// TIA Portal V20 export
VAR_GLOBAL   // PLC tag table "Inputs"
   "Switch 1 ON" AT %I16.0 : Bool;
   "Switch 2 ON" AT %I16.1 : Bool;
   "Switch 3 ON" AT %I16.2 : Bool;
   "Switch 4 ON" AT %I16.3 : Bool;
   "Switch 5 ON" AT %I16.4 : Bool;
   "Switch 6 ON" AT %I16.5 : Bool;
   "Switch 7 ON" AT %I16.6 : Bool;
   "Switch 8 ON" AT %I16.7 : Bool;
   "Byte 1 ON" AT %IB1 : Byte;
   Here_is_a_word AT %IW2 : Word;
END_VAR
